// TIA Portal V20 export
VAR_GLOBAL   // PLC tag table "MABS"
   "MABS_C1.2.1_IN" AT %I100.0 : "IB_P01/02/03_in_64bytes_struct";
   "MABS_C1.2.1_Out" AT %I200.0 : "IB_P01/02/03_out_64bytes_struct";
   "MABS_C1.2.2_IN" AT %I300.0 : "IB_P01/02/03_in_64bytes_struct";
   "MABS_C1.2.2_Out" AT %I400.0 : "IB_P01/02/03_out_64bytes_struct";
END_VAR
